// Mitsubishi GX Works2 project: NOR   PLC: Q03UDV

PROGRAM MAIN
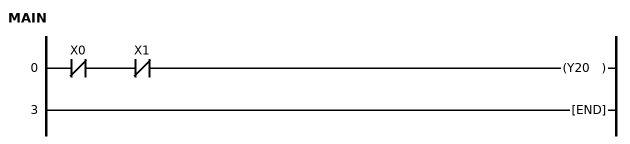
0     LDI     X0
      ANI     X1
      OUT     Y20
3     END
END_PROGRAM
